INTERFACE I_XtsTransport_Mover

METHOD Disable : E_PROGRESS
VAR_INPUT
  Execute             : BOOL;
END_VAR
END_METHOD

METHOD Enable : E_PROGRESS
VAR_INPUT
  Execute             : BOOL;
END_VAR
END_METHOD

METHOD GearIn : E_PROGRESS;
VAR_INPUT
  Execute             : BOOL;
  stMoveData          : ST_MOVE_DATA;
  stGearData          : ST_GEAR_DATA;
END_VAR
END_METHOD

METHOD GearInPosCa : E_PROGRESS
VAR_INPUT
  Execute             : BOOL;
  stMoveData          : ST_MOVE_DATA;
  stGearData          : ST_GEAR_DATA;  
END_VAR
END_METHOD

METHOD GearOut : E_PROGRESS
VAR_INPUT
  Execute             : BOOL;
END_VAR
END_METHOD

METHOD Halt : E_PROGRESS
VAR_INPUT
  Execute             : BOOL;
  stMoveData          : ST_MOVE_DATA;
END_VAR
END_METHOD

PROPERTY MessageLevel : e_messagetype
SET
END_SET
END_PROPERTY

PROPERTY ModuloTurn : dint
GET
END_GET
END_PROPERTY

METHOD MoveToPos : E_PROGRESS
VAR_INPUT
  Execute             : BOOL;
  stMoveData          : ST_MOVE_DATA;
END_VAR
END_METHOD

METHOD MoveToPosCa : E_PROGRESS
VAR_INPUT
  Execute             : BOOL;
  stMoveData          : ST_MOVE_DATA;
END_VAR
END_METHOD

PROPERTY RailLength : LREAL
GET
END_GET
SET
END_SET
END_PROPERTY

METHOD Reset : E_PROGRESS
VAR_INPUT
  Execute             : BOOL;
END_VAR
END_METHOD

METHOD SendToAbsPosCa : E_PROGRESS
VAR_INPUT
  Execute             : BOOL;
  stMoveData          : ST_MOVE_DATA;
END_VAR
END_METHOD

METHOD SendToModuloPosCa : E_PROGRESS
VAR_INPUT
  Execute             : BOOL;
  stMoveData          : ST_MOVE_DATA;
END_VAR
END_METHOD

END_INTERFACE

(* stored: Version 1.1.0.1, ProductVersion 3.1.4024.13
   Itf I_XtsTransport_Mover: Id {6ee03612-2ff4-4a59-90cf-9b7f02d97d43}
   Folder methods: Id {30a78529-75eb-4ec3-b260-b4d9869bc548}
   Folder properties: Id {d070d651-e59b-43e8-938f-2e7a4e773730}
   Method Disable: Id {bbb4094d-4abf-43a0-a4d4-fdb591095cb9}
   Method Enable: Id {5ca3fb26-c3e5-4801-8976-7e308b56585f}
   Method GearIn: Id {aef6abc5-9bb7-4812-bdd7-ca3d79b2f014}
   Method GearInPosCa: Id {4226561b-17a2-4036-b33a-0771a942deda}
   Method GearOut: Id {3fce0a8f-0e77-4639-a8f7-0ecccef8d7f0}
   Method Halt: Id {d32a7df8-de7e-44ef-b6ee-1ec36ad20986}
   Property MessageLevel: Id {e8bc9c50-b4c2-42fc-9f7b-68ba5ba5dc3b}
   Set Set: Id {d13e3888-0345-47d3-aa29-c81d583c63ae}
   Property ModuloTurn: Id {c3977c7f-e42f-4881-a59f-bc880186086f}
   Get Get: Id {80341b40-853e-4fd0-940b-5271fd8fe014}
   Method MoveToPos: Id {b0817eff-ede5-4380-9332-c555330f6e82}
   Method MoveToPosCa: Id {57d96c93-aa0c-4263-be31-4b7c4f7ed139}
   Property RailLength: Id {2ab9a517-e9c4-4297-9032-25295569fe63}
   Get Get: Id {e1ecafed-c266-4265-964e-19044948e250}
   Set Set: Id {6f118226-d1ae-4dcf-be6c-c57da7ca0402}
   Method Reset: Id {17f8812c-28c6-4bd5-9f16-b47ea1a6ae27}
   Method SendToAbsPosCa: Id {e17ec937-1fe5-42b1-a767-8a67b7116d3c}
   Method SendToModuloPosCa: Id {2a99547a-abc5-40b9-8a74-a8d336d66959} *)
